Universal Robots PolyScope program: _adminCG-ConveyorToPHome.urp

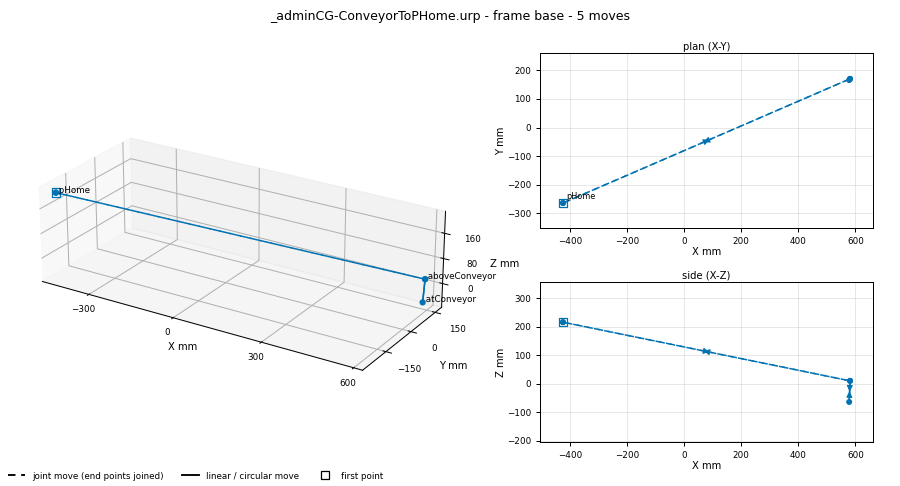
[picture p0: tool path of _adminCG-ConveyorToPHome.urp in frame base, 5 of 5 moves have a stored position in this frame; points joined in program order, loops and branches not executed]
Program _adminCG-ConveyorToPHome (installation=admin directory=/programs/THU_530PM createdIn=3.8.0.61336 lastSavedIn=3.15.8.106339 robotSerialNumber=2015350925)
Calibrated DH parameters: a=[0, -0.425, -0.39225, 0, 0, 0]; d=[0.089159, 0, 0, 0.10915, 0.09465, 0.0823]; alpha=[1.570796, 0, 0, 1.570796, -1.570796, 0]; deltaTheta=[0, 0, 0, 0, 0, 0]
Robot Program (runOnlyOnce=true)
  Set DigitalOutput pin=digital_out[0]; digitalValue=0
  Call _adminLinearIndex1
  MoveJ speed 60 deg/s, acceleration 80 deg/s^2 (useActiveTCP=true)
    Waypoint pHome: TCP in base x=-424.168 y=-264.274 z=215.857 mm, rx=-1.1973 ry=-2.8917 rz=-0.0084 rad; joints [224.995, -90.007, -90.005, -90.014, 89.257, -0.02] deg; flange x=-422.259 y=-266.324 z=431.739 mm, rx=-1.1973 ry=-2.8917 rz=-0.0084 rad
    Waypoint aboveConveyor: TCP in base x=580.867 y=170.525 z=10.509 mm, rx=2.903 ry=-1.1997 rz=-0.0021 rad; joints [26.728, -110.87, -96.027, -63.175, 90.04, -18.366] deg; flange x=581.178 y=170.512 z=226.408 mm, rx=2.903 ry=-1.1997 rz=-0.0021 rad
  MoveL speed 250 mm/s, acceleration 1200 mm/s^2 (useActiveTCP=true) feature=Base
    Waypoint atConveyor: TCP in base x=577.856 y=166.297 z=-63.417 mm, rx=2.9037 ry=-1.1992 rz=-0.0028 rad; joints [26.475, -115.745, -101.44, -52.884, 90.075, -18.645] deg; flange x=578.218 y=166.16 z=152.482 mm, rx=2.9037 ry=-1.1992 rz=-0.0028 rad
    Set DigitalOutput pin=digital_out[0]; digitalValue=1
    Wait Sleep waitTime=1
    Waypoint aboveConveyor: TCP in base x=580.867 y=170.525 z=10.509 mm, rx=2.903 ry=-1.1997 rz=-0.0021 rad; joints [26.728, -110.87, -96.027, -63.175, 90.04, -18.366] deg; flange x=581.178 y=170.512 z=226.408 mm, rx=2.903 ry=-1.1997 rz=-0.0021 rad
  MoveJ speed 60 deg/s, acceleration 80 deg/s^2 (useActiveTCP=true)
    Waypoint pHome: TCP in base x=-424.168 y=-264.274 z=215.857 mm, rx=-1.1973 ry=-2.8917 rz=-0.0084 rad; joints [224.995, -90.007, -90.005, -90.014, 89.257, -0.02] deg; flange x=-422.259 y=-266.324 z=431.739 mm, rx=-1.1973 ry=-2.8917 rz=-0.0084 rad
SubProgram  [hidden by the author, left out]
SubProgram _adminLinearIndex1 [hidden by the author, left out]
